PROGRAM SimpleSafetyProgram
VAR

	fromTwinSafe_GroupInRun AT %I* : BOOL;
	
	toTwinSafe_ResetGroup AT %Q* : BOOL;
	toTwinSafe_StartGroup AT %Q* : BOOL;
	
	toTwinSafe_ResetSafetyProgram AT %Q* : BOOL;	

END_VAR

END_PROGRAM

(* stored: Version 1.1.0.1, ProductVersion 3.1.4024.14
   POU SimpleSafetyProgram: Id {451f3921-d055-4805-a882-c98f3c7f1b11}, SpecialFunc None *)
